// TIA Portal project "ASIT TANKI OTOMASYON UYGULMASI( COMPARATORS 1)" (V18)

(* hardware
DEVICE "S7-1200 station_1"  S7-1200 Station
   slot 0: "Rack_0"  S7-1200 Rack  Rack  V1.0
   slot 1: "PLC_1"  CPU 1214C DC/DC/Rly  6ES7 214-1HG40-0XB0  V4.6
*)

// ===== PLC "PLC_1"  CPU 1214C DC/DC/Rly =====

VAR_GLOBAL   // PLC tag table "Default tag table"
   "START BUT" AT %I0.0 : Bool;
   "STOP BUT" AT %I0.1 : Bool;
   "ACIL STOP BUT" AT %I0.2 : Bool;
   "KARISTIRICI 1" AT %Q0.0 : Bool;
   "KARISTIRICI 2" AT %Q0.1 : Bool;
   "BOSALTMA MOTORU 1" AT %Q0.2 : Bool;
   "BOSALTMA MOTORU 2" AT %Q0.3 : Bool;
   "SISTEM-MEM" AT %M5.0 : Bool;
   "ZAMAN DEGERI" AT %MD50 : Time;
   "SISTEM BASA AL" AT %M5.1 : Bool;
END_VAR

// folder: System blocks/Program resources

DATA_BLOCK "TIMER 1"   // DB1
{ S7_Optimized_Access := 'TRUE' }
AUTHOR : Simatic
FAMILY : IEC
NAME : IEC_TMR
VERSION : 1.0
// stored: InstanceOfName IEC_TIMER
"IEC_TIMER"
BEGIN
END_DATA_BLOCK

// folder: (top level)

ORGANIZATION_BLOCK "Main"   // OB1, LAD, ProgramCycle
TITLE = "Main Program Sweep (Cycle)"
{ S7_Optimized_Access := 'TRUE' }
VERSION : 0.1
   VAR_INPUT
      Initial_Call : Bool;   // Initial call of this OB
      Remanence : Bool;   // =True, if remanent data are available
   END_VAR
   VAR_TEMP   // added for the SCL form of the ladder/FBD networks
      _w1 : Bool;
   END_VAR
BEGIN

REGION Network 1: SİSTEM START / STOP KONTROLÜ
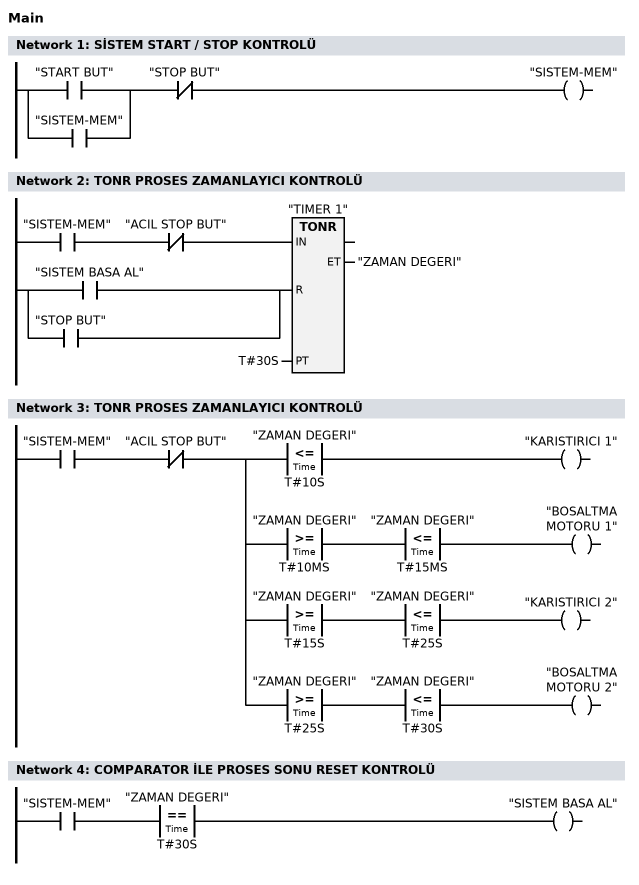
   RUNG wire#powerrail
      Contact( "START BUT" )
      wire#w1
      I_Contact( "STOP BUT" )
      Coil( "SISTEM-MEM" )
   END_RUNG
   RUNG wire#powerrail
      Contact( "SISTEM-MEM" )
   END_RUNG wire#w1
   // the same network as SCL:
   "SISTEM-MEM" := ("START BUT" OR "SISTEM-MEM") AND NOT "STOP BUT";
END_REGION

REGION Network 2: TONR PROSES ZAMANLAYICI KONTROLÜ
   "TIMER 1".TONR(IN := "SISTEM-MEM" AND NOT "ACIL STOP BUT",
                  R := "SISTEM BASA AL" OR "STOP BUT",
                  PT := T#30S,
                  ET => "ZAMAN DEGERI");
END_REGION

REGION Network 3: TONR PROSES ZAMANLAYICI KONTROLÜ
   RUNG wire#powerrail
      Contact( "SISTEM-MEM" )
      I_Contact( "ACIL STOP BUT" )
      wire#w1
      { S7_Templates := "SrcType := Time" } LE_Contact(in1 := "ZAMAN DEGERI", in2 := T#10S)
      Coil( "KARISTIRICI 1" )
   END_RUNG
   RUNG wire#w1
      { S7_Templates := "SrcType := Time" } GE_Contact(in1 := "ZAMAN DEGERI", in2 := T#10MS)
      { S7_Templates := "SrcType := Time" } LE_Contact(in1 := "ZAMAN DEGERI", in2 := T#15MS)
      Coil( "BOSALTMA MOTORU 1" )
   END_RUNG
   RUNG wire#w1
      { S7_Templates := "SrcType := Time" } GE_Contact(in1 := "ZAMAN DEGERI", in2 := T#15S)
      { S7_Templates := "SrcType := Time" } LE_Contact(in1 := "ZAMAN DEGERI", in2 := T#25S)
      Coil( "KARISTIRICI 2" )
   END_RUNG
   RUNG wire#w1
      { S7_Templates := "SrcType := Time" } GE_Contact(in1 := "ZAMAN DEGERI", in2 := T#25S)
      { S7_Templates := "SrcType := Time" } LE_Contact(in1 := "ZAMAN DEGERI", in2 := T#30S)
      Coil( "BOSALTMA MOTORU 2" )
   END_RUNG
   // the same network as SCL:
   #_w1 := "SISTEM-MEM" AND NOT "ACIL STOP BUT";
   "KARISTIRICI 1" := #_w1 AND ("ZAMAN DEGERI" <= T#10S);
   "BOSALTMA MOTORU 1" := #_w1 AND ("ZAMAN DEGERI" >= T#10MS) AND ("ZAMAN DEGERI" <= T#15MS);
   "KARISTIRICI 2" := #_w1 AND ("ZAMAN DEGERI" >= T#15S) AND ("ZAMAN DEGERI" <= T#25S);
   "BOSALTMA MOTORU 2" := #_w1 AND ("ZAMAN DEGERI" >= T#25S) AND ("ZAMAN DEGERI" <= T#30S);
END_REGION

REGION Network 4: COMPARATOR İLE PROSES SONU RESET KONTROLÜ
   RUNG wire#powerrail
      Contact( "SISTEM-MEM" )
      { S7_Templates := "SrcType := Time" } EQ_Contact(in1 := "ZAMAN DEGERI", in2 := T#30S)
      Coil( "SISTEM BASA AL" )
   END_RUNG
   // the same network as SCL:
   "SISTEM BASA AL" := "SISTEM-MEM" AND ("ZAMAN DEGERI" = T#30S);
END_REGION
END_ORGANIZATION_BLOCK